// 隐含生成代码：不要编辑
FUNCTION CheckDivLReal : LREAL
VAR_INPUT
	divisor:LREAL;
END_VAR

// 隐含生成代码：这里只是对代码实现的建议
{noflow}
IF divisor = 0 THEN
	CheckDivLReal:=1;
ELSE
	CheckDivLReal:=divisor;
END_IF;
{flow}

END_FUNCTION

(* stored: Version 1.1.0.1, ProductVersion 3.1.4022.16
   POU CheckDivLReal: Id {aba9ccf4-1a0c-4efa-a767-a951bc41d3f5}, SpecialFunc CheckDivReal64 *)
